// TIA Portal V19 export
FUNCTION_BLOCK "F_Zone27_FB"   // FB170, F_LAD
TITLE = SAFETY ZONE 27 - AREA 03 (CREAZIONE PACCO)
// stored: Access Published
   VAR
      F_Sinamics_SpallaTesta : "FDevice_Sinamics_FB";
      F_Sinamics_SpallaCoda : "FDevice_Sinamics_FB";
      F_Sinamics_TraslazioneTesta : "FDevice_Sinamics_FB";
      F_Sinamics_TraslazioneCoda : "FDevice_Sinamics_FB";
      F_Sinamics_SollevamentoTesta : "FDevice_Sinamics_FB";
      F_Sinamics_SollevamentoCoda : "FDevice_Sinamics_FB";
      F_Sinamics_SostegnoAntiribTesta : "FDevice_Sinamics_FB";
      F_Sinamics_SostegnoAntiribCoda : "FDevice_Sinamics_FB";
      F_SafetyValve_Air_A0302_A0303 : "FDevice_Valve_FB";
   END_VAR
   VAR_TEMP
      DoorNormalStop : Bool;
      DoorSafeStop : Bool;
      Door_Ok : Bool;
      FDBK : Bool;
   END_VAR
BEGIN

REGION Network 1: < < < < < < < < < < DOOR > > > > > > > > > >
END_REGION

REGION Network 2: -
END_REGION

REGION Network 3: < < < < < < < < < < ZONE SAFETY INTERFACE > > > > > > > > > >
END_REGION

REGION Network 4: Cumulative Zone Safety
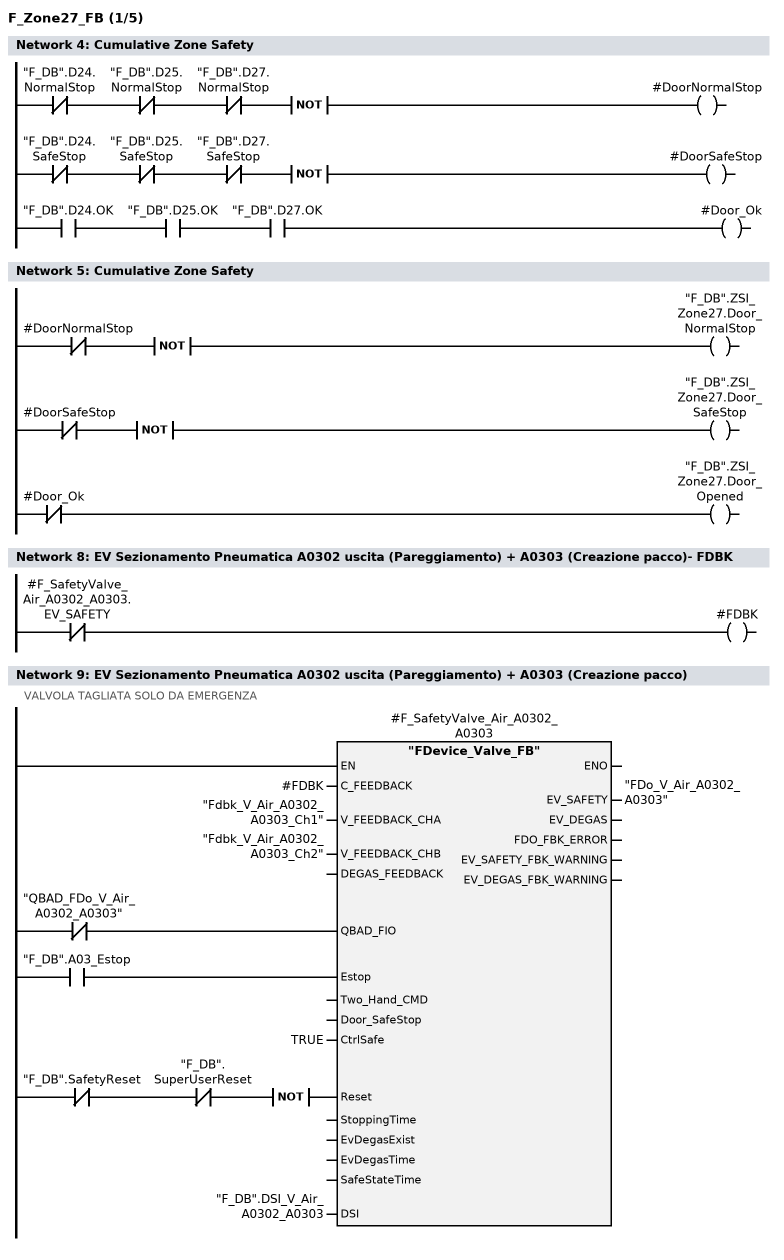
   RUNG wire#powerrail
      I_Contact( "F_DB".D24.NormalStop )
      I_Contact( "F_DB".D25.NormalStop )
      I_Contact( "F_DB".D27.NormalStop )
      Not()
      Coil( #DoorNormalStop )
   END_RUNG
   RUNG wire#powerrail
      I_Contact( "F_DB".D24.SafeStop )
      I_Contact( "F_DB".D25.SafeStop )
      I_Contact( "F_DB".D27.SafeStop )
      Not()
      Coil( #DoorSafeStop )
   END_RUNG
   RUNG wire#powerrail
      Contact( "F_DB".D24.OK )
      Contact( "F_DB".D25.OK )
      Contact( "F_DB".D27.OK )
      Coil( #Door_Ok )
   END_RUNG
   // the same network as SCL:
   #DoorNormalStop := NOT (NOT "F_DB".D24.NormalStop AND NOT "F_DB".D25.NormalStop AND NOT "F_DB".D27.NormalStop);
   #DoorSafeStop := NOT (NOT "F_DB".D24.SafeStop AND NOT "F_DB".D25.SafeStop AND NOT "F_DB".D27.SafeStop);
   #Door_Ok := "F_DB".D24.OK AND "F_DB".D25.OK AND "F_DB".D27.OK;
END_REGION

REGION Network 5: Cumulative Zone Safety
   RUNG wire#powerrail
      I_Contact( #DoorNormalStop )
      Not()
      Coil( "F_DB".ZSI_Zone27.Door_NormalStop )
   END_RUNG
   RUNG wire#powerrail
      I_Contact( #DoorSafeStop )
      Not()
      Coil( "F_DB".ZSI_Zone27.Door_SafeStop )
   END_RUNG
   RUNG wire#powerrail
      I_Contact( #Door_Ok )
      Coil( "F_DB".ZSI_Zone27.Door_Opened )
   END_RUNG
   // the same network as SCL:
   "F_DB".ZSI_Zone27.Door_NormalStop := NOT (NOT #DoorNormalStop);
   "F_DB".ZSI_Zone27.Door_SafeStop := NOT (NOT #DoorSafeStop);
   "F_DB".ZSI_Zone27.Door_Opened := NOT #Door_Ok;
END_REGION

REGION Network 6: >
END_REGION

REGION Network 7: < < < < < < < < < < DEVICES SAFETY VALVES > > > > > > > > > >
END_REGION

REGION Network 8: EV Sezionamento Pneumatica A0302 uscita (Pareggiamento) + A0303 (Creazione pacco)- FDBK
   RUNG wire#powerrail
      I_Contact( #F_SafetyValve_Air_A0302_A0303.EV_SAFETY )
      Coil( #FDBK )
   END_RUNG
   // the same network as SCL:
   #FDBK := NOT #F_SafetyValve_Air_A0302_A0303.EV_SAFETY;
END_REGION

REGION Network 9: EV Sezionamento Pneumatica A0302 uscita (Pareggiamento) + A0303 (Creazione pacco)
   // VALVOLA TAGLIATA SOLO DA EMERGENZA
   RUNG wire#powerrail
      #F_SafetyValve_Air_A0302_A0303(QBAD_FIO := wire#w1, Estop := wire#w2, Reset := wire#w3, C_FEEDBACK := #FDBK, V_FEEDBACK_CHA := "Fdbk_V_Air_A0302_A0303_Ch1", V_FEEDBACK_CHB := "Fdbk_V_Air_A0302_A0303_Ch2", DEGAS_FEEDBACK :=, Two_Hand_CMD :=, Door_SafeStop :=, CtrlSafe := TRUE, StoppingTime :=, EvDegasExist :=, EvDegasTime :=, SafeStateTime :=, DSI := "F_DB".DSI_V_Air_A0302_A0303, EV_SAFETY => "FDo_V_Air_A0302_A0303", EV_DEGAS =>, FDO_FBK_ERROR =>, EV_SAFETY_FBK_WARNING =>, EV_DEGAS_FBK_WARNING =>)
   END_RUNG
   RUNG wire#powerrail
      I_Contact( "QBAD_FDo_V_Air_A0302_A0303" )
   END_RUNG wire#w1
   RUNG wire#powerrail
      Contact( "F_DB".A03_Estop )
   END_RUNG wire#w2
   RUNG wire#powerrail
      I_Contact( "F_DB".SafetyReset )
      I_Contact( "F_DB".SuperUserReset )
      Not()
   END_RUNG wire#w3
   // the same network as SCL:
   #F_SafetyValve_Air_A0302_A0303(C_FEEDBACK := #FDBK,   // "FDevice_Valve_FB"
                           V_FEEDBACK_CHA := "Fdbk_V_Air_A0302_A0303_Ch1",
                           V_FEEDBACK_CHB := "Fdbk_V_Air_A0302_A0303_Ch2",
                           QBAD_FIO := NOT "QBAD_FDo_V_Air_A0302_A0303",
                           Estop := "F_DB".A03_Estop,
                           CtrlSafe := TRUE,
                           Reset := NOT (NOT "F_DB".SafetyReset AND NOT "F_DB".SuperUserReset),
                           DSI := "F_DB".DSI_V_Air_A0302_A0303,
                           EV_SAFETY => "FDo_V_Air_A0302_A0303");
END_REGION

REGION Network 11: >
END_REGION

REGION Network 12: < < < < < < < < < < DEVICES CONTACTORS > > > > > > > > > >
END_REGION

REGION Network 13: >
END_REGION

REGION Network 14: < < < < < < < < < < DEVICES S120 > > > > > > > > > >
END_REGION

REGION Network 15: S120 - Ax Spalla Testa
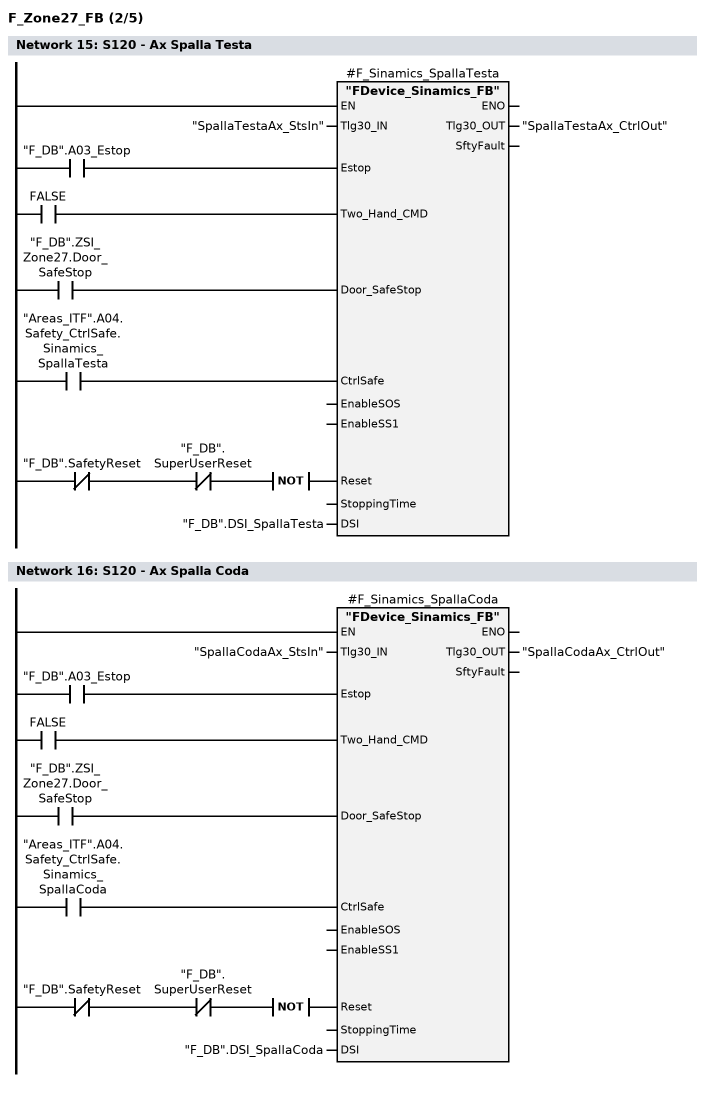
   RUNG wire#powerrail
      #F_Sinamics_SpallaTesta(Estop := wire#w1, Two_Hand_CMD := wire#w2, Door_SafeStop := wire#w3, CtrlSafe := wire#w4, Reset := wire#w5, Tlg30_IN := "SpallaTestaAx_StsIn", EnableSOS :=, EnableSS1 :=, StoppingTime :=, DSI := "F_DB".DSI_SpallaTesta, Tlg30_OUT => "SpallaTestaAx_CtrlOut", SftyFault =>)
   END_RUNG
   RUNG wire#powerrail
      Contact( "F_DB".A03_Estop )
   END_RUNG wire#w1
   RUNG wire#powerrail
      Contact( FALSE )
   END_RUNG wire#w2
   RUNG wire#powerrail
      Contact( "F_DB".ZSI_Zone27.Door_SafeStop )
   END_RUNG wire#w3
   RUNG wire#powerrail
      Contact( "Areas_ITF".A04.Safety_CtrlSafe.Sinamics_SpallaTesta )
   END_RUNG wire#w4
   RUNG wire#powerrail
      I_Contact( "F_DB".SafetyReset )
      I_Contact( "F_DB".SuperUserReset )
      Not()
   END_RUNG wire#w5
   // the same network as SCL:
   #F_Sinamics_SpallaTesta(Tlg30_IN := "SpallaTestaAx_StsIn",   // "FDevice_Sinamics_FB"
                           Estop := "F_DB".A03_Estop,
                           Two_Hand_CMD := FALSE,
                           Door_SafeStop := "F_DB".ZSI_Zone27.Door_SafeStop,
                           CtrlSafe := "Areas_ITF".A04.Safety_CtrlSafe.Sinamics_SpallaTesta,
                           Reset := NOT (NOT "F_DB".SafetyReset AND NOT "F_DB".SuperUserReset),
                           DSI := "F_DB".DSI_SpallaTesta,
                           Tlg30_OUT => "SpallaTestaAx_CtrlOut");
END_REGION

REGION Network 16: S120 - Ax Spalla Coda
   RUNG wire#powerrail
      #F_Sinamics_SpallaCoda(Estop := wire#w1, Two_Hand_CMD := wire#w2, Door_SafeStop := wire#w3, CtrlSafe := wire#w4, Reset := wire#w5, Tlg30_IN := "SpallaCodaAx_StsIn", EnableSOS :=, EnableSS1 :=, StoppingTime :=, DSI := "F_DB".DSI_SpallaCoda, Tlg30_OUT => "SpallaCodaAx_CtrlOut", SftyFault =>)
   END_RUNG
   RUNG wire#powerrail
      Contact( "F_DB".A03_Estop )
   END_RUNG wire#w1
   RUNG wire#powerrail
      Contact( FALSE )
   END_RUNG wire#w2
   RUNG wire#powerrail
      Contact( "F_DB".ZSI_Zone27.Door_SafeStop )
   END_RUNG wire#w3
   RUNG wire#powerrail
      Contact( "Areas_ITF".A04.Safety_CtrlSafe.Sinamics_SpallaCoda )
   END_RUNG wire#w4
   RUNG wire#powerrail
      I_Contact( "F_DB".SafetyReset )
      I_Contact( "F_DB".SuperUserReset )
      Not()
   END_RUNG wire#w5
   // the same network as SCL:
   #F_Sinamics_SpallaCoda(Tlg30_IN := "SpallaCodaAx_StsIn",   // "FDevice_Sinamics_FB"
                          Estop := "F_DB".A03_Estop,
                          Two_Hand_CMD := FALSE,
                          Door_SafeStop := "F_DB".ZSI_Zone27.Door_SafeStop,
                          CtrlSafe := "Areas_ITF".A04.Safety_CtrlSafe.Sinamics_SpallaCoda,
                          Reset := NOT (NOT "F_DB".SafetyReset AND NOT "F_DB".SuperUserReset),
                          DSI := "F_DB".DSI_SpallaCoda,
                          Tlg30_OUT => "SpallaCodaAx_CtrlOut");
END_REGION

REGION Network 17: S120 - Ax Traslazione Testa
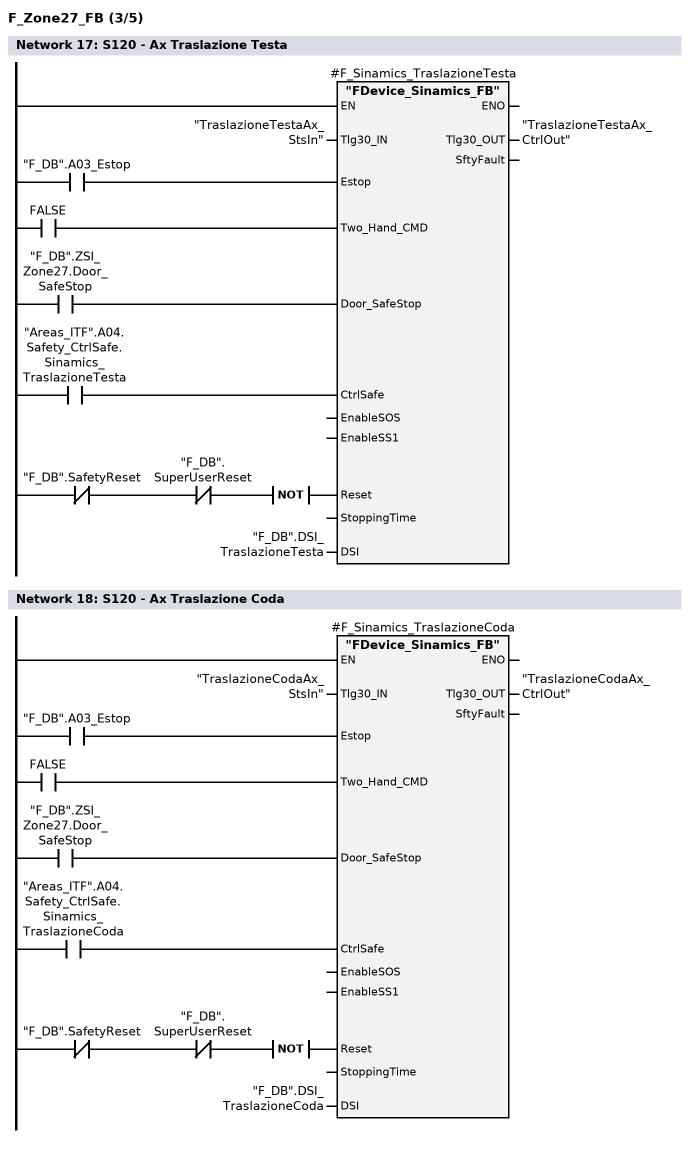
   RUNG wire#powerrail
      #F_Sinamics_TraslazioneTesta(Estop := wire#w1, Two_Hand_CMD := wire#w2, Door_SafeStop := wire#w3, CtrlSafe := wire#w4, Reset := wire#w5, Tlg30_IN := "TraslazioneTestaAx_StsIn", EnableSOS :=, EnableSS1 :=, StoppingTime :=, DSI := "F_DB".DSI_TraslazioneTesta, Tlg30_OUT => "TraslazioneTestaAx_CtrlOut", SftyFault =>)
   END_RUNG
   RUNG wire#powerrail
      Contact( "F_DB".A03_Estop )
   END_RUNG wire#w1
   RUNG wire#powerrail
      Contact( FALSE )
   END_RUNG wire#w2
   RUNG wire#powerrail
      Contact( "F_DB".ZSI_Zone27.Door_SafeStop )
   END_RUNG wire#w3
   RUNG wire#powerrail
      Contact( "Areas_ITF".A04.Safety_CtrlSafe.Sinamics_TraslazioneTesta )
   END_RUNG wire#w4
   RUNG wire#powerrail
      I_Contact( "F_DB".SafetyReset )
      I_Contact( "F_DB".SuperUserReset )
      Not()
   END_RUNG wire#w5
   // the same network as SCL:
   #F_Sinamics_TraslazioneTesta(Tlg30_IN := "TraslazioneTestaAx_StsIn",   // "FDevice_Sinamics_FB"
                           Estop := "F_DB".A03_Estop,
                           Two_Hand_CMD := FALSE,
                           Door_SafeStop := "F_DB".ZSI_Zone27.Door_SafeStop,
                           CtrlSafe := "Areas_ITF".A04.Safety_CtrlSafe.Sinamics_TraslazioneTesta,
                           Reset := NOT (NOT "F_DB".SafetyReset AND NOT "F_DB".SuperUserReset),
                           DSI := "F_DB".DSI_TraslazioneTesta,
                           Tlg30_OUT => "TraslazioneTestaAx_CtrlOut");
END_REGION

REGION Network 18: S120 - Ax Traslazione Coda
   RUNG wire#powerrail
      #F_Sinamics_TraslazioneCoda(Estop := wire#w1, Two_Hand_CMD := wire#w2, Door_SafeStop := wire#w3, CtrlSafe := wire#w4, Reset := wire#w5, Tlg30_IN := "TraslazioneCodaAx_StsIn", EnableSOS :=, EnableSS1 :=, StoppingTime :=, DSI := "F_DB".DSI_TraslazioneCoda, Tlg30_OUT => "TraslazioneCodaAx_CtrlOut", SftyFault =>)
   END_RUNG
   RUNG wire#powerrail
      Contact( "F_DB".A03_Estop )
   END_RUNG wire#w1
   RUNG wire#powerrail
      Contact( FALSE )
   END_RUNG wire#w2
   RUNG wire#powerrail
      Contact( "F_DB".ZSI_Zone27.Door_SafeStop )
   END_RUNG wire#w3
   RUNG wire#powerrail
      Contact( "Areas_ITF".A04.Safety_CtrlSafe.Sinamics_TraslazioneCoda )
   END_RUNG wire#w4
   RUNG wire#powerrail
      I_Contact( "F_DB".SafetyReset )
      I_Contact( "F_DB".SuperUserReset )
      Not()
   END_RUNG wire#w5
   // the same network as SCL:
   #F_Sinamics_TraslazioneCoda(Tlg30_IN := "TraslazioneCodaAx_StsIn",   // "FDevice_Sinamics_FB"
                           Estop := "F_DB".A03_Estop,
                           Two_Hand_CMD := FALSE,
                           Door_SafeStop := "F_DB".ZSI_Zone27.Door_SafeStop,
                           CtrlSafe := "Areas_ITF".A04.Safety_CtrlSafe.Sinamics_TraslazioneCoda,
                           Reset := NOT (NOT "F_DB".SafetyReset AND NOT "F_DB".SuperUserReset),
                           DSI := "F_DB".DSI_TraslazioneCoda,
                           Tlg30_OUT => "TraslazioneCodaAx_CtrlOut");
END_REGION

REGION Network 19: S120 - Ax Sollevamento Testa
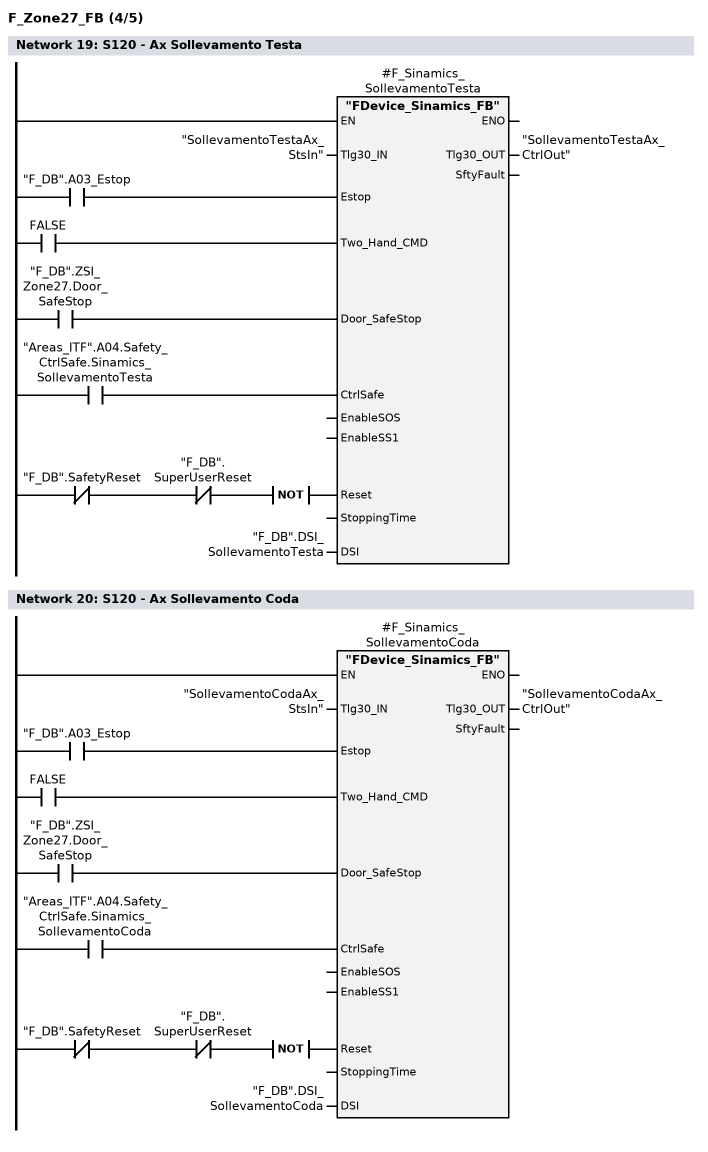
   RUNG wire#powerrail
      #F_Sinamics_SollevamentoTesta(Estop := wire#w1, Two_Hand_CMD := wire#w2, Door_SafeStop := wire#w3, CtrlSafe := wire#w4, Reset := wire#w5, Tlg30_IN := "SollevamentoTestaAx_StsIn", EnableSOS :=, EnableSS1 :=, StoppingTime :=, DSI := "F_DB".DSI_SollevamentoTesta, Tlg30_OUT => "SollevamentoTestaAx_CtrlOut", SftyFault =>)
   END_RUNG
   RUNG wire#powerrail
      Contact( "F_DB".A03_Estop )
   END_RUNG wire#w1
   RUNG wire#powerrail
      Contact( FALSE )
   END_RUNG wire#w2
   RUNG wire#powerrail
      Contact( "F_DB".ZSI_Zone27.Door_SafeStop )
   END_RUNG wire#w3
   RUNG wire#powerrail
      Contact( "Areas_ITF".A04.Safety_CtrlSafe.Sinamics_SollevamentoTesta )
   END_RUNG wire#w4
   RUNG wire#powerrail
      I_Contact( "F_DB".SafetyReset )
      I_Contact( "F_DB".SuperUserReset )
      Not()
   END_RUNG wire#w5
   // the same network as SCL:
   #F_Sinamics_SollevamentoTesta(Tlg30_IN := "SollevamentoTestaAx_StsIn",   // "FDevice_Sinamics_FB"
                           Estop := "F_DB".A03_Estop,
                           Two_Hand_CMD := FALSE,
                           Door_SafeStop := "F_DB".ZSI_Zone27.Door_SafeStop,
                           CtrlSafe := "Areas_ITF".A04.Safety_CtrlSafe.Sinamics_SollevamentoTesta,
                           Reset := NOT (NOT "F_DB".SafetyReset AND NOT "F_DB".SuperUserReset),
                           DSI := "F_DB".DSI_SollevamentoTesta,
                           Tlg30_OUT => "SollevamentoTestaAx_CtrlOut");
END_REGION

REGION Network 20: S120 - Ax Sollevamento Coda
   RUNG wire#powerrail
      #F_Sinamics_SollevamentoCoda(Estop := wire#w1, Two_Hand_CMD := wire#w2, Door_SafeStop := wire#w3, CtrlSafe := wire#w4, Reset := wire#w5, Tlg30_IN := "SollevamentoCodaAx_StsIn", EnableSOS :=, EnableSS1 :=, StoppingTime :=, DSI := "F_DB".DSI_SollevamentoCoda, Tlg30_OUT => "SollevamentoCodaAx_CtrlOut", SftyFault =>)
   END_RUNG
   RUNG wire#powerrail
      Contact( "F_DB".A03_Estop )
   END_RUNG wire#w1
   RUNG wire#powerrail
      Contact( FALSE )
   END_RUNG wire#w2
   RUNG wire#powerrail
      Contact( "F_DB".ZSI_Zone27.Door_SafeStop )
   END_RUNG wire#w3
   RUNG wire#powerrail
      Contact( "Areas_ITF".A04.Safety_CtrlSafe.Sinamics_SollevamentoCoda )
   END_RUNG wire#w4
   RUNG wire#powerrail
      I_Contact( "F_DB".SafetyReset )
      I_Contact( "F_DB".SuperUserReset )
      Not()
   END_RUNG wire#w5
   // the same network as SCL:
   #F_Sinamics_SollevamentoCoda(Tlg30_IN := "SollevamentoCodaAx_StsIn",   // "FDevice_Sinamics_FB"
                           Estop := "F_DB".A03_Estop,
                           Two_Hand_CMD := FALSE,
                           Door_SafeStop := "F_DB".ZSI_Zone27.Door_SafeStop,
                           CtrlSafe := "Areas_ITF".A04.Safety_CtrlSafe.Sinamics_SollevamentoCoda,
                           Reset := NOT (NOT "F_DB".SafetyReset AND NOT "F_DB".SuperUserReset),
                           DSI := "F_DB".DSI_SollevamentoCoda,
                           Tlg30_OUT => "SollevamentoCodaAx_CtrlOut");
END_REGION

REGION Network 21: S120 - Ax Sostegno Antiribaltamento Testa
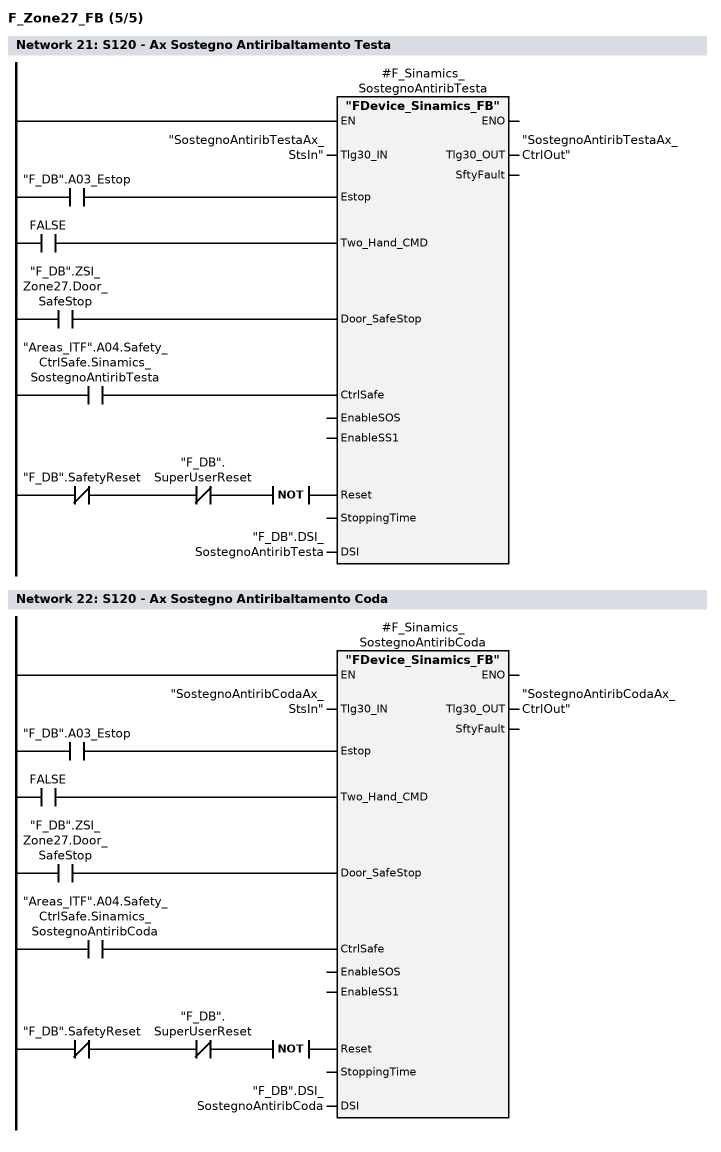
   RUNG wire#powerrail
      #F_Sinamics_SostegnoAntiribTesta(Estop := wire#w1, Two_Hand_CMD := wire#w2, Door_SafeStop := wire#w3, CtrlSafe := wire#w4, Reset := wire#w5, Tlg30_IN := "SostegnoAntiribTestaAx_StsIn", EnableSOS :=, EnableSS1 :=, StoppingTime :=, DSI := "F_DB".DSI_SostegnoAntiribTesta, Tlg30_OUT => "SostegnoAntiribTestaAx_CtrlOut", SftyFault =>)
   END_RUNG
   RUNG wire#powerrail
      Contact( "F_DB".A03_Estop )
   END_RUNG wire#w1
   RUNG wire#powerrail
      Contact( FALSE )
   END_RUNG wire#w2
   RUNG wire#powerrail
      Contact( "F_DB".ZSI_Zone27.Door_SafeStop )
   END_RUNG wire#w3
   RUNG wire#powerrail
      Contact( "Areas_ITF".A04.Safety_CtrlSafe.Sinamics_SostegnoAntiribTesta )
   END_RUNG wire#w4
   RUNG wire#powerrail
      I_Contact( "F_DB".SafetyReset )
      I_Contact( "F_DB".SuperUserReset )
      Not()
   END_RUNG wire#w5
   // the same network as SCL:
   #F_Sinamics_SostegnoAntiribTesta(Tlg30_IN := "SostegnoAntiribTestaAx_StsIn",   // "FDevice_Sinamics_FB"
                           Estop := "F_DB".A03_Estop,
                           Two_Hand_CMD := FALSE,
                           Door_SafeStop := "F_DB".ZSI_Zone27.Door_SafeStop,
                           CtrlSafe := "Areas_ITF".A04.Safety_CtrlSafe.Sinamics_SostegnoAntiribTesta,
                           Reset := NOT (NOT "F_DB".SafetyReset AND NOT "F_DB".SuperUserReset),
                           DSI := "F_DB".DSI_SostegnoAntiribTesta,
                           Tlg30_OUT => "SostegnoAntiribTestaAx_CtrlOut");
END_REGION

REGION Network 22: S120 - Ax Sostegno Antiribaltamento Coda
   RUNG wire#powerrail
      #F_Sinamics_SostegnoAntiribCoda(Estop := wire#w1, Two_Hand_CMD := wire#w2, Door_SafeStop := wire#w3, CtrlSafe := wire#w4, Reset := wire#w5, Tlg30_IN := "SostegnoAntiribCodaAx_StsIn", EnableSOS :=, EnableSS1 :=, StoppingTime :=, DSI := "F_DB".DSI_SostegnoAntiribCoda, Tlg30_OUT => "SostegnoAntiribCodaAx_CtrlOut", SftyFault =>)
   END_RUNG
   RUNG wire#powerrail
      Contact( "F_DB".A03_Estop )
   END_RUNG wire#w1
   RUNG wire#powerrail
      Contact( FALSE )
   END_RUNG wire#w2
   RUNG wire#powerrail
      Contact( "F_DB".ZSI_Zone27.Door_SafeStop )
   END_RUNG wire#w3
   RUNG wire#powerrail
      Contact( "Areas_ITF".A04.Safety_CtrlSafe.Sinamics_SostegnoAntiribCoda )
   END_RUNG wire#w4
   RUNG wire#powerrail
      I_Contact( "F_DB".SafetyReset )
      I_Contact( "F_DB".SuperUserReset )
      Not()
   END_RUNG wire#w5
   // the same network as SCL:
   #F_Sinamics_SostegnoAntiribCoda(Tlg30_IN := "SostegnoAntiribCodaAx_StsIn",   // "FDevice_Sinamics_FB"
                           Estop := "F_DB".A03_Estop,
                           Two_Hand_CMD := FALSE,
                           Door_SafeStop := "F_DB".ZSI_Zone27.Door_SafeStop,
                           CtrlSafe := "Areas_ITF".A04.Safety_CtrlSafe.Sinamics_SostegnoAntiribCoda,
                           Reset := NOT (NOT "F_DB".SafetyReset AND NOT "F_DB".SuperUserReset),
                           DSI := "F_DB".DSI_SostegnoAntiribCoda,
                           Tlg30_OUT => "SostegnoAntiribCodaAx_CtrlOut");
END_REGION

REGION Network 23: >
END_REGION

REGION Network 24: >
END_REGION
END_FUNCTION_BLOCK
